(****************************************************************************************)
(*							Beckhoff Automation Poland									*)
(*							L_TBConvByteToBits     v1.0									*)
(*									29.02.2007											*)
(*	This FB returns the 8 corresponding bit values for an input value of type ”byte”	*)
(*______________________________________________________________________________________*)
FUNCTION_BLOCK L_TBConvByteToBits
VAR_INPUT
	byInput: BYTE;
END_VAR
VAR_OUTPUT
	bBit0: BOOL;
	bBit1: BOOL;
	bBit2: BOOL;
	bBit3: BOOL;
	bBit4: BOOL;
	bBit5: BOOL;
	bBit6: BOOL;
	bBit7: BOOL;
END_VAR

bBit0 := byInput.0;
bBit1 := byInput.1;
bBit2 := byInput.2;
bBit3 := byInput.3;
bBit4 := byInput.4;
bBit5 := byInput.5;
bBit6 := byInput.6;
bBit7 := byInput.7;

END_FUNCTION_BLOCK

(* stored: Version 1.1.0.1, ProductVersion 3.1.4026.13, FileIdentifier 512afe3c3eb4df4151917f3f616f5d42bee70252, FileSignature 3c0c5d9f479dd06c171f96f42f0f9cd7c06c04d71c877eded28493c2eeaeed6d55c278aca17291d7854e7096595112a372359024117588798cc946598fdb908febe5b23b3a7a7aca54db8ec92e6ca087e4dc95d45cc0f8ec8dad71a3114e0cc6d31c136edf45a0c7f25d049031878a6d90200960a9c07cf72b63ae4d79eadfd0e7e90eb4bb8d10fa57e800b42995582e466fbdb38c7ec598c72048ce58ce78e0b06d5c4b67005fc26a486dac8bf4f38c00d94bb84ed03915e851d29e871acca0dd934514d4defcebc7936eed63280d049b71783975739e98edf64833a8aa01765e99089f970b549e3e762da27627c6b28fbef4d190d9491ac34f4455f7e424da
   POU L_TBConvByteToBits: Id {74296ea7-7e10-4bb2-80d2-b7313a7dfc0b}, SpecialFunc None *)
